TYPE DUT_PARAMETER_INPUT :
STRUCT
	///Value of the parameter 
	Value: LREAL;
	///Possibility to a string value depending on the parameter
	StringValue: STRING[80];
END_STRUCT
END_TYPE

(* stored: Version 1.1.0.1, ProductVersion 3.1.0.25
   DUT DUT_PARAMETER_INPUT: Id {cb111b7c-09f7-4b07-9270-2a07e3509831} *)
